PROGRAM Inicio
VAR
	Premarcha: BOOL;
	TmrPremarcha: TON;
END_VAR
VAR // added by the converter: edge detectors and wires of the graphical bodies
    _rt1 : R_TRIG;
    _w1, _w2 : BOOL;
END_VAR

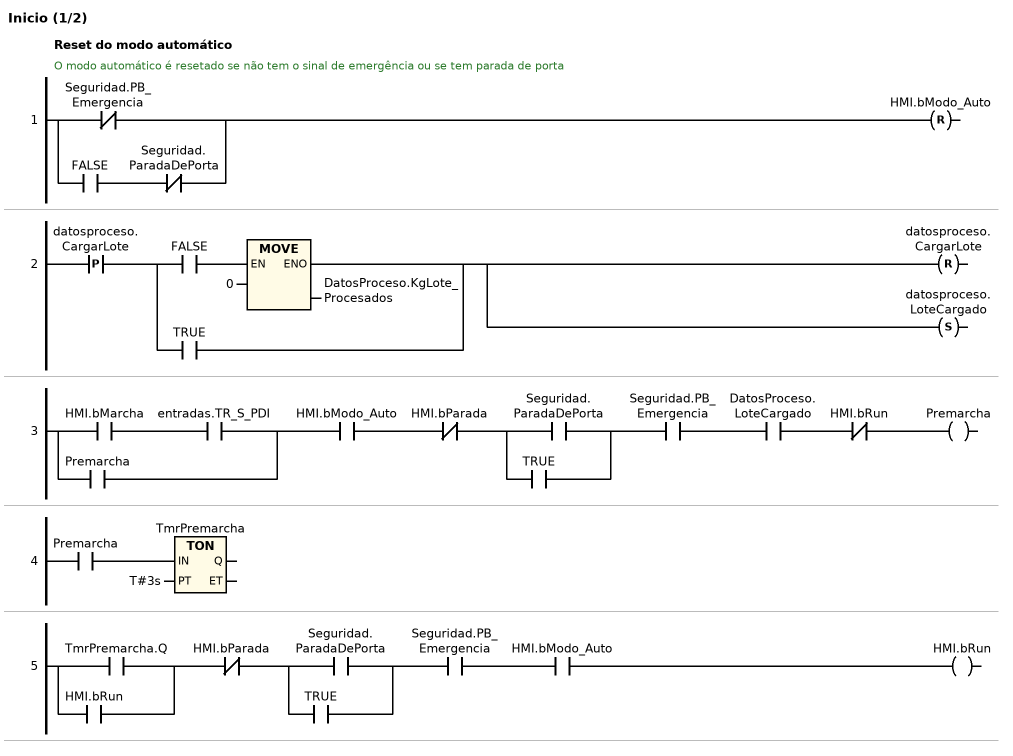
// NETWORK 1: Reset do modo automático
// O modo automático é resetado se não tem o sinal de emergência ou se tem parada de porta
HMI.bModo_Auto R= NOT Seguridad.PB_Emergencia OR FALSE AND NOT Seguridad.ParadaDePorta;

// NETWORK 2
_rt1(CLK := datosproceso.CargarLote);
_w1 := _rt1.Q AND TRUE;
IF NOT _w1 THEN
    _w2 := _rt1.Q AND FALSE;
    IF _w2 THEN DatosProceso.KgLote_Procesados := 0; END_IF
    _w1 := _w2;
END_IF
datosproceso.CargarLote R= _w1;
datosproceso.LoteCargado S= _w1;

// NETWORK 3
Premarcha := (HMI.bMarcha AND entradas.TR_S_PDI OR Premarcha) AND HMI.bModo_Auto AND NOT HMI.bParada AND (Seguridad.ParadaDePorta OR TRUE) AND Seguridad.PB_Emergencia AND DatosProceso.LoteCargado AND NOT HMI.bRun;

// NETWORK 4
TmrPremarcha(IN := Premarcha, PT := T#3s); // TON

// NETWORK 5
HMI.bRun := (TmrPremarcha.Q OR HMI.bRun) AND NOT HMI.bParada AND (Seguridad.ParadaDePorta OR TRUE) AND Seguridad.PB_Emergencia AND HMI.bModo_Auto;

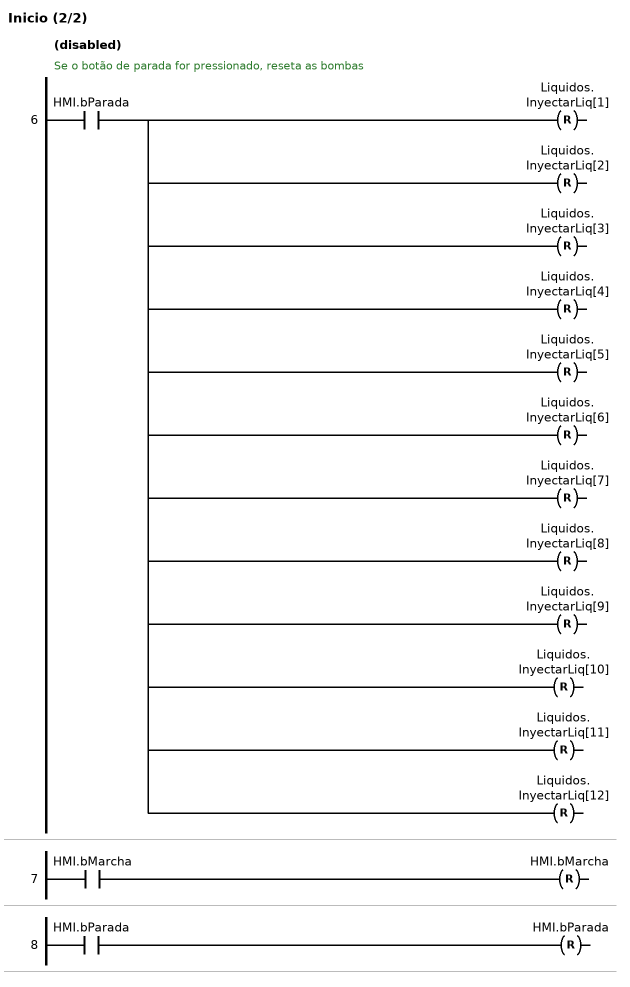
// NETWORK 6 (disabled)
// Se o botão de parada for pressionado, reseta as bombas
// Liquidos.InyectarLiq[1] R= HMI.bParada;
// Liquidos.InyectarLiq[2] R= HMI.bParada;
// Liquidos.InyectarLiq[3] R= HMI.bParada;
// Liquidos.InyectarLiq[4] R= HMI.bParada;
// Liquidos.InyectarLiq[5] R= HMI.bParada;
// Liquidos.InyectarLiq[6] R= HMI.bParada;
// Liquidos.InyectarLiq[7] R= HMI.bParada;
// Liquidos.InyectarLiq[8] R= HMI.bParada;
// Liquidos.InyectarLiq[9] R= HMI.bParada;
// Liquidos.InyectarLiq[10] R= HMI.bParada;
// Liquidos.InyectarLiq[11] R= HMI.bParada;
// Liquidos.InyectarLiq[12] R= HMI.bParada;

// NETWORK 7
HMI.bMarcha R= HMI.bMarcha;

// NETWORK 8
HMI.bParada R= HMI.bParada;

END_PROGRAM

(* stored: Version 1.1.0.1, ProductVersion 3.1.4024.14
   POU Inicio: Id {0475ed7c-2281-44cd-bcf3-046e46b1536c}, SpecialFunc None *)
